FUNCTION_BLOCK FB_ACTION
VAR_INPUT
	sNAME: STRING;
	PIST: REFERENCE TO FB_PISTON;
	aLIFT:REFERENCE TO FB_Axis;
	aXY:REFERENCE TO FB_Axis;
	bSTART_OPEN:BOOL;
	bSTART_CLOSE:BOOL;
	bSTART_HOMING:BOOL;
	iHOME_STATE:INT:=98;
	iOPEN_STATE:INT:=98;
	iCLOSE_STATE:INT:=98;
	bHOME_ALL:BOOL;
	bOPEN_ALL:BOOL;
	bCLOSE_ALL:BOOL;
	tACTION:TON;
	rACTION_TIMEOUT:TIME:=T#20S;
	tHOMING:TON;
	rHOMING_TIMEOUT: TIME:=T#20S;
	tOPEN:TON;
	rOPEN_TIMEOUT: TIME:=T#20S;
	tCLOSE:TON;
	rCLOSE_TIMEOUT: TIME:=T#20S;
END_VAR
VAR_OUTPUT
	sACTION_STATE:STRING:='UNINIT';
	bSTART_ACTION:BOOL;
	iACTION_STATE:INT:=98;
	bACTION_ERROR:BOOL;
	bALL_HOMED:BOOL;
	bALL_OPENED:BOOL;
	bALL_CLOSED:BOOL;
END_VAR
VAR
END_VAR

mACTION_STATE_MACHINE();
IF bALL_HOMED THEN
	IF NOT aLIFT.bHOMED OR NOT aXY.bHOMED THEN
		bALL_HOMED:=FALSE;
		iACTION_STATE:=98;
	END_IF
END_IF

ACTION aACTION_ERROR:
gEventType:= 'action Alarm'; 
gEventSeverity:= 'Error';

gEventName:= sNAME;
IF iACTION_STATE=2  THEN
	gEventText:='action XY homing';
	gEventIdentity:=5001;
END_IF
IF iACTION_STATE=2  THEN
	gEventText:='action LIFT homing';
	gEventIdentity:=5002;
END_IF
IF iACTION_STATE=5  THEN
	gEventText:='action PISTON homing';
	gEventIdentity:=5003;
END_IF
//---------------------------------------------------
IF iACTION_STATE=14  THEN
	gEventText:='action XY opening';
	gEventIdentity:=5011;
END_IF
IF iACTION_STATE=12  THEN
	gEventText:='action LIFT opening';
	gEventIdentity:=5012;
END_IF
IF iACTION_STATE=10  THEN
	gEventText:='action PISTON opening';
	gEventIdentity:=5013;
END_IF
//---------------------------------------------------
IF iACTION_STATE=32  THEN
	gEventText:='action XY closing';
	gEventIdentity:=5021;
END_IF
IF iACTION_STATE=34  THEN
	gEventText:='action LIFT closing';
	gEventIdentity:=5022;
END_IF
IF iACTION_STATE=35  THEN
	gEventText:='action PISTON closing';
	gEventIdentity:=5023;
END_IF
fbEventLogger.mAdd();
END_ACTION

METHOD mACTION_STATE_MACHINE : BOOL
VAR_INPUT
END_VAR
 tACTION(IN:= bSTART_ACTION, PT:=rACTION_TIMEOUT , Q=> , ET=> );

CASE iACTION_STATE OF
	
	1://======================================  HOME ALL	
		//HOME XY
		sACTION_STATE:='HOMING ALL XY';
		bHOME_ALL:=FALSE; bALL_HOMED:=FALSE;bALL_OPENED:=FALSE;bOPEN_ALL:=FALSE;bALL_CLOSED:=FALSE;bCLOSE_ALL:=FALSE;
		aXY.bHome:=TRUE;
		bSTART_ACTION:=TRUE;
		iACTION_STATE:=2; 
	2:
		aXY.bHome:=FALSE;
		IF aXY.bHOMED THEN
			bSTART_ACTION:=FALSE;
			iACTION_STATE:=3;
		END_IF
		IF aXY.bSTATE_ERROR THEN
			iACTION_STATE:=99;
			aACTION_ERROR();
			bSTART_ACTION:=FALSE;
			bACTION_ERROR:=TRUE;
		END_IF
			
	3://HOME LIFT
		sACTION_STATE:='HOMING ALL LIFT';
		aLIFT.bHome:=TRUE;
		bSTART_ACTION:=TRUE;
		iACTION_STATE:=4;
	4:
		aLIFT.bHome:=FALSE;
		IF aLIFT.bHOMED THEN
			bSTART_ACTION:=FALSE;
			iACTION_STATE:=5;
		END_IF
		IF aLIFT.bSTATE_ERROR THEN
			aACTION_ERROR();
			iACTION_STATE:=99;
			bSTART_ACTION:=FALSE;
			bACTION_ERROR:=TRUE;
		END_IF
	5://HOME PISTON
		sACTION_STATE:='HOMING ALL PISTON';
		bSTART_ACTION:=TRUE;
		PIST.bOPEN_SWR:=FALSE;
		IF PIST.bCLOSED THEN
			bSTART_ACTION:=FALSE;
			iACTION_STATE:=100;
			bALL_HOMED:=TRUE;
		END_IF
		IF PIST.bERROR THEN
			aACTION_ERROR();
			iACTION_STATE:=99;
			bSTART_ACTION:=FALSE;
			bACTION_ERROR:=TRUE;
		END_IF
	10://===================================== OPENING ALL
		//OPEN PISTON
		bHOME_ALL:=FALSE; bALL_HOMED:=FALSE;bALL_OPENED:=FALSE;bOPEN_ALL:=FALSE;bALL_CLOSED:=FALSE;bCLOSE_ALL:=FALSE;
		sACTION_STATE:='OPENING ALL PISTON';
		bSTART_ACTION:=TRUE;
		PIST.bOPEN_SWR:=TRUE;
		IF PIST.bOPENED THEN
			bSTART_ACTION:=FALSE;
			iACTION_STATE:=11;
		END_IF
		IF PIST.bERROR THEN
			aACTION_ERROR();
			iACTION_STATE:=99;
			bSTART_ACTION:=FALSE;
			bACTION_ERROR:=TRUE;
		END_IF
	11://OPEN LIFT
		sACTION_STATE:='OPENING ALL LIFT';
		aLIFT.bOPEN:=TRUE;
		bSTART_ACTION:=TRUE;
		iACTION_STATE:=12;
	12:
		aLIFT.bOPEN:=FALSE;
		IF aLIFT.bOPENED THEN
			bSTART_ACTION:=FALSE;
			iACTION_STATE:=13;
		END_IF
		IF aLIFT.bSTATE_ERROR THEN
			aACTION_ERROR();
			iACTION_STATE:=99;
			bSTART_ACTION:=FALSE;
			bACTION_ERROR:=TRUE;
		END_IF
	13://OPEN ALL XY
		sACTION_STATE:='OPENING ALL XY';
		aXY.bOPEN:=TRUE;
		bSTART_ACTION:=TRUE;
		iACTION_STATE:=14; 
	14:
		aXY.bOPEN:=FALSE;
		IF aXY.bOPENED THEN
			bSTART_ACTION:=FALSE;
			bALL_OPENED:=TRUE;
			iACTION_STATE:=20;
		END_IF
		IF aXY.bSTATE_ERROR THEN
			aACTION_ERROR();
			iACTION_STATE:=99;
			bSTART_ACTION:=FALSE;
			bACTION_ERROR:=TRUE;
		END_IF	

	20:// ==================================== OPENED
		sACTION_STATE:='OPENED';
		IF bCLOSE_ALL THEN
			iACTION_STATE:=30;
			bACTION_ERROR:=FALSE;
		END_IF
		IF bHOME_ALL THEN
			iACTION_STATE:=1;
			bACTION_ERROR:=FALSE;
		END_IF
		
	30://===================================== CLOSING ALL XY
		sACTION_STATE:='CLOSING ALL XY';
		bHOME_ALL:=FALSE; bALL_HOMED:=FALSE;bALL_OPENED:=FALSE;bOPEN_ALL:=FALSE;bALL_CLOSED:=FALSE;bCLOSE_ALL:=FALSE;
		aXY.bCLOSE:=TRUE;
		bSTART_ACTION:=TRUE;
		iACTION_STATE:=32; 
	32:
		aXY.bCLOSE:=FALSE;
		IF aXY.bCLOSED THEN
			bSTART_ACTION:=FALSE;
			iACTION_STATE:=33;
		END_IF
		IF aXY.bSTATE_ERROR THEN
			aACTION_ERROR();
			iACTION_STATE:=99;
			bSTART_ACTION:=FALSE;
			bACTION_ERROR:=TRUE;
		END_IF	
	33://HOME LIFT
		sACTION_STATE:='CLOSING ALL LIFT';
		aLIFT.bCLOSE:=TRUE;
		bSTART_ACTION:=TRUE;
		iACTION_STATE:=34;
	34:
		aLIFT.bCLOSE:=FALSE;
		IF aLIFT.bCLOSED THEN
			bSTART_ACTION:=FALSE;
			iACTION_STATE:=35;
		END_IF
		IF aLIFT.bSTATE_ERROR THEN
			aACTION_ERROR();
			iACTION_STATE:=99;
			bSTART_ACTION:=FALSE;
			bACTION_ERROR:=TRUE;
		END_IF
	35://CLOSE ALL PISTON
		sACTION_STATE:='CLOSING ALL PISTON';
		bSTART_ACTION:=TRUE;
		PIST.bOPEN_SWR:=FALSE;
		IF PIST.bCLOSED THEN
			bSTART_ACTION:=FALSE;
			iACTION_STATE:=40;
			bALL_CLOSED:=TRUE;
		END_IF
		IF PIST.bERROR THEN
			aACTION_ERROR();
			iACTION_STATE:=99;
			bSTART_ACTION:=FALSE;
			bACTION_ERROR:=TRUE;
		END_IF 
	40:// ==================================== CLOSED
		sACTION_STATE:='CLOSED';
		IF bOPEN_ALL THEN
			iACTION_STATE:=10;
			bACTION_ERROR:=FALSE;
		END_IF		
		IF bHOME_ALL THEN
			iACTION_STATE:=1;
			bACTION_ERROR:=FALSE;
		END_IF
		
	98://===================================== UNINIT
		sACTION_STATE:='UNINIT';
		IF bHOME_ALL THEN
			iACTION_STATE:=1;
			bACTION_ERROR:=FALSE;
		END_IF
		
	99://===================================== ERROR
		sACTION_STATE:='ERROR';
		IF bHOME_ALL THEN
			iACTION_STATE:=1;
			bACTION_ERROR:=FALSE;
		END_IF
	
	100://===================================== HOMED
		sACTION_STATE:='HOMED';
		IF bHOME_ALL THEN
			iACTION_STATE:=1;
			bACTION_ERROR:=FALSE;
		END_IF	
		IF bOPEN_ALL THEN
			iACTION_STATE:=10;
			bACTION_ERROR:=FALSE;
		END_IF
	
	
END_CASE
END_METHOD

END_FUNCTION_BLOCK

(* stored: Version 1.1.0.1, ProductVersion 3.1.4024.12
   POU FB_ACTION: Id {77b4196e-a6d2-4735-ae2e-ed59e88b663e}, SpecialFunc None
   Action aACTION_ERROR: Id {18ded634-2282-4c0c-b5aa-75bbf974bd96}
   Method mACTION_STATE_MACHINE: Id {3aea7e34-a6ec-43c3-a03c-1c552f7c93cb} *)
